Fanuc KAREL source: kd00052.KL

-- PROVISIONAL review KL for V940-1; original PC SHA256 f1d2b3ffcad519836486d01d8ba7170ed834d622cbcc4e00671bbc60c35a7825
-- Incomplete behavior may be omitted. Consult companion uncertainty JSON. Do not deploy.
PROGRAM KD00052
%NOLOCKGROUP
VAR
  I : INTEGER
  J : INTEGER
  B : BOOLEAN
  R : REAL
  S : STRING[80]
-- UNRESOLVED_DECL P type=000101
BEGIN
  -- V9_ZERO_TABLE_METADATA_HINT layout=0001; no indexed target words; source/name/runtime held
  -- UNRESOLVED_PC offsets 5-42; opcodes 01,22,1C,06,82,03,9D,2E,51,9D,12,9D,1B,9D,13,04,0B
  -- UNRESOLVED_PC offsets 47-51; opcodes 7F
END KD00052
